FUNCTION_BLOCK DrillingContainer EXTENDS ZCore.ObjectContainer
VAR_INPUT
END_VAR
VAR_OUTPUT
END_VAR
VAR
  {attribute 'hide'}
  _parent : REFERENCE TO DrillingUnit;
END_VAR

{ attribute 'hide' }
METHOD FB_init : BOOL
VAR_INPUT
	bInitRetains : BOOL; // if TRUE, the retain variables are initialized (warm start / cold start)
	bInCopyCode : BOOL;  // if TRUE, the instance afterwards gets moved into the copy code (online change)
  unit : REFERENCE TO DrillingUnit;
END_VAR
_parent REF= unit;
END_METHOD

END_FUNCTION_BLOCK

(* stored: Version 1.1.0.1
   POU DrillingContainer: Id {30cf670d-92da-40f3-8509-6b36eaf93e94}, SpecialFunc None
   Method FB_init: Id {c0be20b2-502b-46f9-8bcb-77e1aafecf1e} *)
